{attribute 'qualified_only'}
VAR_GLOBAL

	Mover			:	ARRAY[0..9] OF AXIS_REF;
	
	Asse_Reale		: Axis_ref;
	Asse_Virtuale	: Axis_ref;

END_VAR

(* stored: Version 1.1.0.1, ProductVersion 3.1.4024.11
   GVL GVL: Id {2637825a-fbfa-4c19-b28f-8bbea4dad5dd} *)
